Omron CX-Programmer project NewProject (CX-Programmer 9.73)

# PLC NewPLC1: CP2E S

## Global symbols (name address type ; comment)
0.00 BOOL  ; input_wlc_cleaning
0.01 BOOL  ; input_wlc_disfect
0.02 BOOL  ; input_wlc_glazing
0.03 BOOL  ; input_thermostat_heater_fan
0.04 BOOL  ; input_thermostat_heater_air
100.00 BOOL  ; relay_pompa_drain
100.01 BOOL  ; relay_pompa_circle
100.02 BOOL  ; relay_clean
100.03 BOOL  ; Relay_disfect
100.04 BOOL  ; relay_glazing
100.05 BOOL  ; relay_hot_fan
100.06 BOOL  ; relay_heater_fan
100.07 BOOL  ; relay_heater_water
101.00 BOOL  ; relay_air_biasa
101.01 BOOL  ; relay_air_bersih
101.02 BOOL  ; relay_lampu_power
101.03 BOOL  ; relay_lampu_runing
101.04 BOOL  ; relay_lampu_error
102 CHANNEL  ; Penambahan_perangkat_analog
2 CHANNEL  ; Pengambilan_data_sensor_suhu
23.00 BOOL  ; perintah_relay_drain
23.01 BOOL  ; perintah_relay_circle
23.02 BOOL  ; perintah_sedot_cleaner
23.03 BOOL  ; perintah_disfect
23.04 BOOL  ; perintah_glazing
23.05 BOOL  ; perintah_hot_fan
23.06 BOOL  ; perintah_heater_water
23.07 BOOL  ; perintah_selenoid_air_kotor
23.08 BOOL  ; relay_selenoid_air_bersih
23.09 BOOL  ; lampu_power
23.10 BOOL  ; perintah_lampu_running
23.11 BOOL  ; perintah_lampu_error
23.13 BOOL  ; perintah_relay_heater_angin
D0 CHANNEL  ; menyimpan_data_sensor
D100 CHANNEL  ; Data sampling
D200 CHANNEL  ; Hasil scalling
D5 CHANNEL  ; Nilai Suhu
T000 BOOL  ; timer_sensor

## Program NewProgram1 (cyclic task 0)

### Section Section1

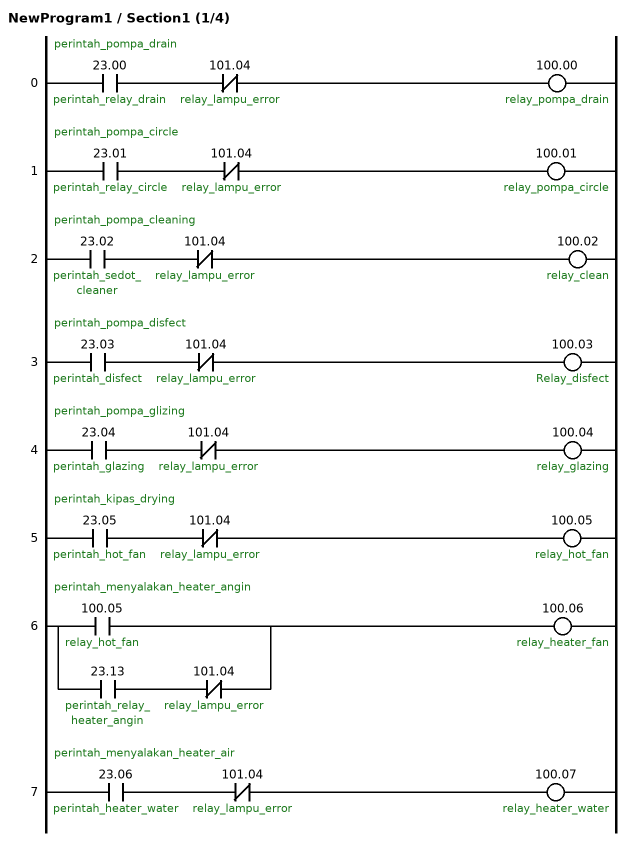
; rung 0: perintah_pompa_drain
LD 23.00  ; perintah_relay_drain
ANDNOT 101.04  ; relay_lampu_error
OUT 100.00  ; relay_pompa_drain
; rung 1: perintah_pompa_circle
LD 23.01  ; perintah_relay_circle
ANDNOT 101.04  ; relay_lampu_error
OUT 100.01  ; relay_pompa_circle
; rung 2: perintah_pompa_cleaning
LD 23.02  ; perintah_sedot_cleaner
ANDNOT 101.04  ; relay_lampu_error
OUT 100.02  ; relay_clean
; rung 3: perintah_pompa_disfect
LD 23.03  ; perintah_disfect
ANDNOT 101.04  ; relay_lampu_error
OUT 100.03  ; Relay_disfect
; rung 4: perintah_pompa_glizing
LD 23.04  ; perintah_glazing
ANDNOT 101.04  ; relay_lampu_error
OUT 100.04  ; relay_glazing
; rung 5: perintah_kipas_drying
LD 23.05  ; perintah_hot_fan
ANDNOT 101.04  ; relay_lampu_error
OUT 100.05  ; relay_hot_fan
; rung 6: perintah_menyalakan_heater_angin
LD 100.05  ; relay_hot_fan
LD 23.13  ; perintah_relay_heater_angin
ANDNOT 101.04  ; relay_lampu_error
ORLD
OUT 100.06  ; relay_heater_fan
; rung 7: perintah_menyalakan_heater_air
LD 23.06  ; perintah_heater_water
ANDNOT 101.04  ; relay_lampu_error
OUT 100.07  ; relay_heater_water

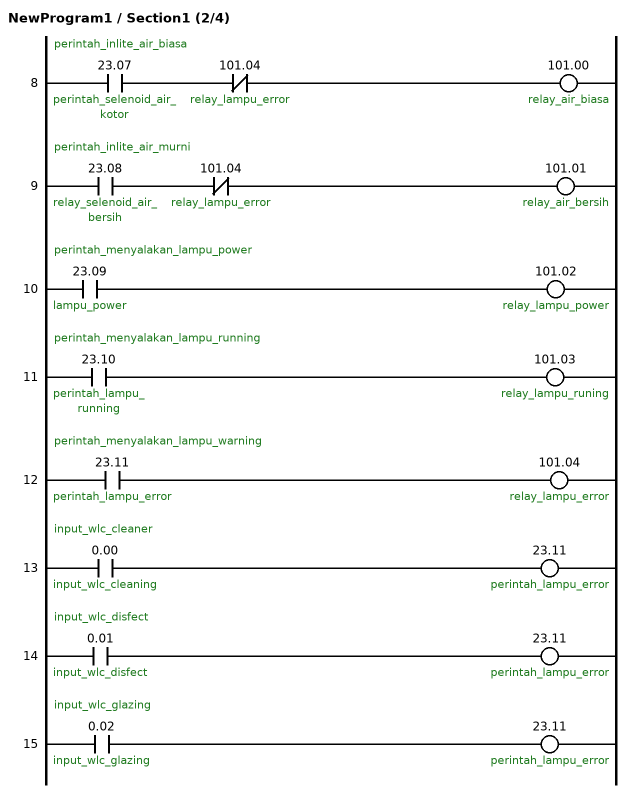
; rung 8: perintah_inlite_air_biasa
LD 23.07  ; perintah_selenoid_air_kotor
ANDNOT 101.04  ; relay_lampu_error
OUT 101.00  ; relay_air_biasa
; rung 9: perintah_inlite_air_murni
LD 23.08  ; relay_selenoid_air_bersih
ANDNOT 101.04  ; relay_lampu_error
OUT 101.01  ; relay_air_bersih
; rung 10: perintah_menyalakan_lampu_power
LD 23.09  ; lampu_power
OUT 101.02  ; relay_lampu_power
; rung 11: perintah_menyalakan_lampu_running
LD 23.10  ; perintah_lampu_running
OUT 101.03  ; relay_lampu_runing
; rung 12: perintah_menyalakan_lampu_warning
LD 23.11  ; perintah_lampu_error
OUT 101.04  ; relay_lampu_error
; rung 13: input_wlc_cleaner
LD 0.00  ; input_wlc_cleaning
OUT 23.11  ; perintah_lampu_error
; rung 14: input_wlc_disfect
LD 0.01  ; input_wlc_disfect
OUT 23.11  ; perintah_lampu_error
; rung 15: input_wlc_glazing
LD 0.02  ; input_wlc_glazing
OUT 23.11  ; perintah_lampu_error

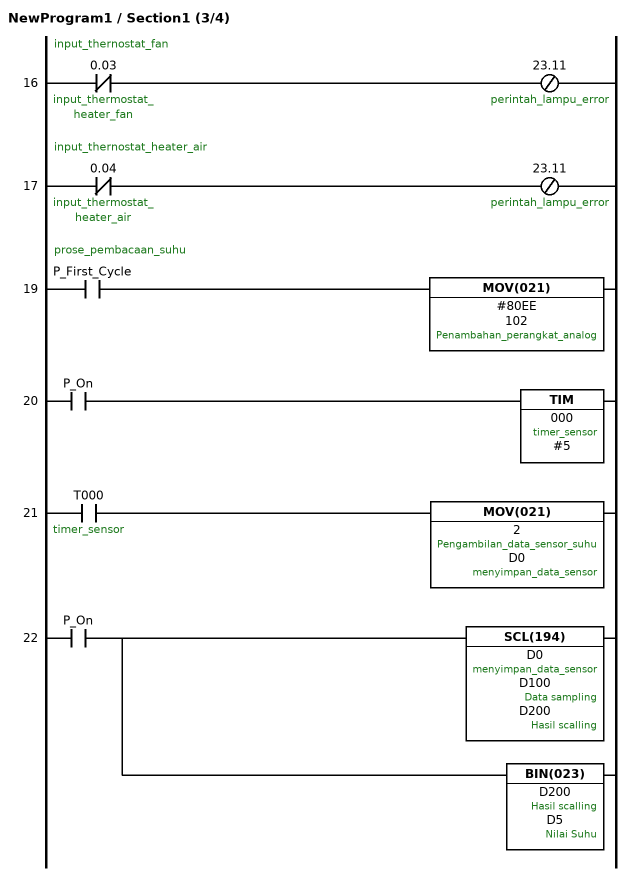
; rung 16: input_thernostat_fan
LDNOT 0.03  ; input_thermostat_heater_fan
OUTNOT 23.11  ; perintah_lampu_error
; rung 17: input_thernostat_heater_air
LDNOT 0.04  ; input_thermostat_heater_air
OUTNOT 23.11  ; perintah_lampu_error
; rung 19: prose_pembacaan_suhu
LD P_First_Cycle
MOV(021) #80EE 102  ; Penambahan_perangkat_analog
; rung 20
LD P_On
TIM 000 #5  ; timer_sensor
; rung 21
LD T000  ; timer_sensor
MOV(021) 2 D0  ; Pengambilan_data_sensor_suhu, menyimpan_data_sensor
; rung 22
LD P_On
SCL(194) D0 D100 D200  ; menyimpan_data_sensor, Data sampling, Hasil scalling
BIN(023) D200 D5  ; Hasil scalling, Nilai Suhu

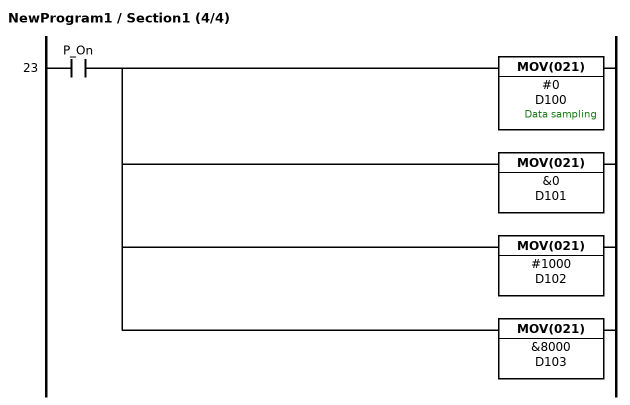
; rung 23
LD P_On
MOV(021) #0 D100  ; Data sampling
MOV(021) &0 D101
MOV(021) #1000 D102
MOV(021) &8000 D103

### Section END
; rung 0
END(001)